// TIA Portal V19 export
DATA_BLOCK "Config"   // DB195
// stored: MemoryReserve 100, Namespace Unit
   VAR
      unit { ExternalWritable := 'False'} : "LAF_typeUnitConfiguration";   // Configuration of Unit Parameters
      stateMachine { ExternalWritable := 'False'} : "LUC_typeStateMachineConfiguration";
      signalStack { ExternalWritable := 'False'} : "LUC_typeSignalStackConfiguration";
      remoteCtrlOpcUa { ExternalWritable := 'False'} : "LUC_typeRemoteCtrlConfiguration";
      stateModeManager { ExternalWritable := 'False'} : "LPMLV2022_typeConfiguration";   // Do not change. Can be configured through stateMachineConfiguration
   END_VAR
BEGIN
   unit.referenceDesignator.relative := WSTRING#'Unit';
END_DATA_BLOCK
